(* CODESYS project Server_02.project

Project tree, tasks and I/O mapping:
  Device : CPX-CEC-C1-V3, Festo AG & Co. KG, order no. 3473128, version 3.5.7.30
      unmapped channels: Rotary switch
    application Application
      libraries: Standard, * (System)
      task MainTask (cyclic, interval t#20ms, priority 20) calls PLC_PRG
      program PLC_PRG [LD]
    PLC_Diagnosis : PLC-Diagnosis, Festo AG & Co. KG, version 3.5.4.1
    CPX_System : CPX_System, Festo AG & Co. KG, order no. 3473128, version 1.233
      CEC_C1_V3 : CEC-C1-V3, Festo AG & Co. KG, order no. 3473128, version 1.233
      _8DI_8DO : 8DI/8DO, Festo AG & Co. KG, order no. 526257, version 1.233
          settings:  = 1;  = 1;  = 1;  = 1;  = 0;  = 1;  = 1;  = 0;  = 0;  = 0;  = 0;  = 0;  = 0;  = 0;  = 0;  = 0;  = 0;  = 0;  = 0;  = 0;  = 0;  = 0;  = 0;  = 0;  = 0;  = 0;  = 0;  = 0;  = 0;  = 0;  = 0;  = 0;  = 0;  = 0;  = 0;  = 0;  = 0;  = 0;  = 0;  = 0;
             = 0;  = 0;  = 0;  = 0;  = 0;  = 0;  = 0;  = 0;  = 0;  = 0;  = 0;  = 0;  = 0;  = 0;  = 0;  = 0;  = 0;  = 0;  = 0;  = 0;  = 0;  = 0;  = 0;  = 0;  = 0;  = 0;  = 0;  = 0;  = 0;  = 0;  = 0;  = 0;  = 0;  = 0;  = 0;  = 0;  = 0;  = 0;  = 0;  = 'PI%i.0.0.1=1';
             = 'PI%i.0.1.1=1';  = 'PI%i.0.2.1=1';  = 'PI%i.1.0.1=1';  = 'PI%i.1.1.1=0';  = 'PI%i.1.4.2=1';  = 'PI%i.1.6.2=1';  = 'PI%i.6.0.1=0';  = 'PI%i.6.1.1=0';  = 'PI%i.6.2.1=0';  = 'PI%i.6.3.1=0';  = 'PI%i.6.4.1=0';  = 'PI%i.6.5.1=0';  = 'PI%i.6.6.1=0';  = 'PI%i.6.7.1=0';  = -;  = -
          input  presenca_peca_inicio : BOOL  // Input 0.Bit0
          input  peca_no_sensor_dist : BOOL  // Input 0.Bit1
          input  sensor_dist : BOOL  // Input 0.Bit2
          input  modulo_desvio_recuado : BOOL  // Input 0.Bit3
          input  sensor_1 : BOOL  // Input 0.Bit4
          input  sensor_2 : BOOL  // Input 0.Bit5
          output esteira_1 : BOOL  // Output 0.Bit0
          output esteira_2 : BOOL  // Output 0.Bit1
          output avanco_cilindrico : BOOL  // Output 0.Bit2
          output avanco_desvio : BOOL  // Output 0.Bit3
          unmapped channels: Input 0, Output 0
      _8DI_8DO_1 : 8DI/8DO, Festo AG & Co. KG, order no. 526257, version 1.233
          unmapped channels: Input 0, Output 0
*)

// Device/Application/PLC_PRG
PROGRAM PLC_PRG
VAR
	presenca_peca_inicioo:BOOL;
	peca_no_sensor_distt:BOOL;
	sensor_distt:BOOL;
	moduo_desvio_recuadoo:BOOL;
	sensor_11:BOOL;
	sensor_22:BOOL;
	
	esteira_11:BOOL;
	esteira_22:BOOL;
	avanco_cilindricoo:BOOL;
	avanco_desvioo:BOOL;
END_VAR

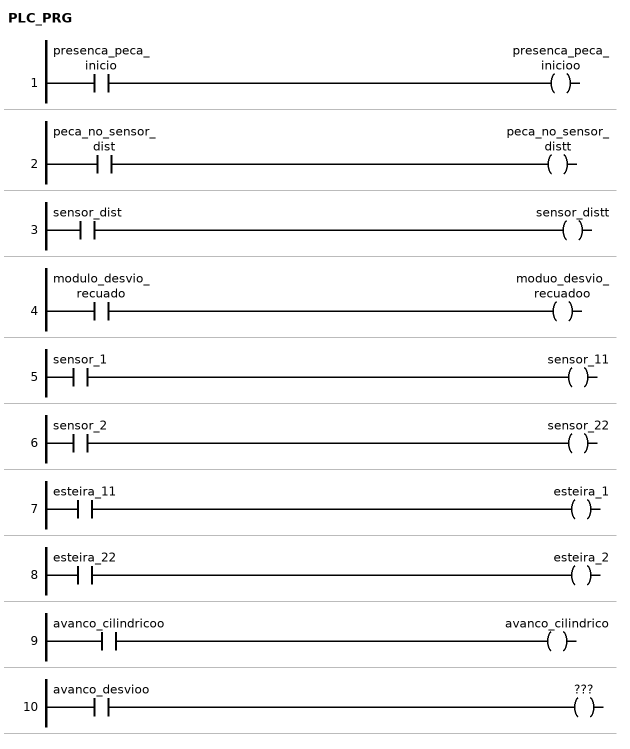
// NETWORK 1
presenca_peca_inicioo := presenca_peca_inicio;

// NETWORK 2
peca_no_sensor_distt := peca_no_sensor_dist;

// NETWORK 3
sensor_distt := sensor_dist;

// NETWORK 4
moduo_desvio_recuadoo := modulo_desvio_recuado;

// NETWORK 5
sensor_11 := sensor_1;

// NETWORK 6
sensor_22 := sensor_2;

// NETWORK 7
esteira_1 := esteira_11;

// NETWORK 8
esteira_2 := esteira_22;

// NETWORK 9
avanco_cilindrico := avanco_cilindricoo;

// NETWORK 10
??? := avanco_desvioo;

END_PROGRAM
